Universal Robots PolyScope program: new.urp

Program new (installation=default directory=/programs/usbdisk/new folder createdIn=5.12.2.1101534 lastSavedIn=5.12.2.1101534 robotSerialNumber=20225202267)
Calibrated DH parameters: a=[0.000057, -0.560337, -0.56987, 0.000044, 0.000023, 0]; d=[0.180974, -304.223407, 295.067386, 9.330269, 0.119831, 0.115671]; alpha=[1.570416, 0.000812, 0.004616, 1.569457, -1.570316, 0]; deltaTheta=[0, -0.415128, 6.624286, 0.074029, 0.000002, -0.000001]
Robot Program (runOnlyOnce=true)
  URCap MigaWeld (Migaweld, Smooth Robotics ApS) dataModel(id_key=0, tag_version=Version1_1, enable_start_button=true, node_defined=true)
    MoveJ speed 60 deg/s, acceleration 80 deg/s^2 (useActiveTCP=false) feature=Base
      Waypoint Home_position: TCP in base x=580.944 y=-683.156 z=684.176 mm, rx=-0.0105 ry=2.8514 rz=-0.1729 rad; joints [-39.068, -105.334, -75.995, -71.646, 95.235, 51.255] deg
    Wait DigitalInput pin=digital_in[1]; digitalValue=1
    SuppressedNode
      Wait DigitalInput pin=digital_in[1]; digitalValue=1
    URCap SpeedSlider (Migaweld, Smooth Robotics ApS) dataModel(set_speed=true)
    SuppressedNode
      URCap WeldParameters (Migaweld, Smooth Robotics ApS) dataModel(processnumber=113, tackWelding=false, duo=false, current=250, isjobselected=true, seqnumber_job=1, puls=true, jobnumber=7)
    SuppressedNode
      Halt
    URCap WeldItem (Migapath, Smooth Robotics ApS) dataModel(MigaPathtitle_key=WeldItem_1)
      URCap Weld seam (Migapath, Smooth Robotics ApS) dataModel(dataModelVersion=1, programVersion=1, travelSpeed=6.0, amplitude=1.4, titleKey=Weld seam, freq=1.5)
        URCap AirPoint (Migapath, Smooth Robotics ApS) dataModel(title_key=Airpoint, jump_visible=true, pose_has_been_offset=false, Pose(key=move_pose_key, Position(key=posePosition, Length(key=X value=0.629812 unit=M), Length(key=Y value=-0.677734 unit=M), Length(key=Z value=0.186771 unit=M)), Rotation(key=poseRotation, Angle(key=RX value=-1.744823 unit=RAD), Angle(key=RY value=1.701375 unit=RAD), Angle(key=RZ value=0.596492 unit=RAD))), JointPositions(key=move_joint_key, JointPosition(key=[1], Angle(key=pos value=-0.681948 unit=RAD)), JointPosition(key=[2], Angle(key=pos value=-1.838358 unit=RAD)), JointPosition(key=[3], Angle(key=pos value=-1.393197 unit=RAD)), JointPosition(key=[4], Angle(key=pos value=-1.363283 unit=RAD)), JointPosition(key=[5], Angle(key=pos value=1.661996 unit=RAD)), JointPosition(key=[6], Angle(key=pos value=0.894606 unit=RAD))))
        URCap AirPoint (Migapath, Smooth Robotics ApS) dataModel(title_key=Startpoint, pose_has_been_offset=false, Pose(key=move_pose_key, Position(key=posePosition, Length(key=X value=0.564215 unit=M), Length(key=Y value=-0.556384 unit=M), Length(key=Z value=0.100836 unit=M)), Rotation(key=poseRotation, Angle(key=RX value=-1.592271 unit=RAD), Angle(key=RY value=1.653557 unit=RAD), Angle(key=RZ value=0.851113 unit=RAD))), JointPositions(key=move_joint_key, JointPosition(key=[1], Angle(key=pos value=-0.675332 unit=RAD)), JointPosition(key=[2], Angle(key=pos value=-1.837109 unit=RAD)), JointPosition(key=[3], Angle(key=pos value=-1.509481 unit=RAD)), JointPosition(key=[4], Angle(key=pos value=-1.463401 unit=RAD)), JointPosition(key=[5], Angle(key=pos value=1.748985 unit=RAD)), JointPosition(key=[6], Angle(key=pos value=0.902886 unit=RAD))))
        URCap Arc On (Migaweld, Smooth Robotics ApS) dataModel(arcOnWaitTime=0.0)
        URCap Paths: (Migapath, Smooth Robotics ApS)
          URCap Welding path (Migapath, Smooth Robotics ApS) dataModel(titleKey=Linear_1, selectedPathType=Linear, useShared=true, selectedPattern=ZigZag, end_has_been_offset=false, Pose(key=endPose, Position(key=posePosition, Length(key=X value=0.594829 unit=M), Length(key=Y value=-0.556361 unit=M), Length(key=Z value=0.100774 unit=M)), Rotation(key=poseRotation, Angle(key=RX value=-1.592161 unit=RAD), Angle(key=RY value=1.653589 unit=RAD), Angle(key=RZ value=0.851163 unit=RAD))), JointPositions(key=endJoint, JointPosition(key=[1], Angle(key=pos value=-0.653154 unit=RAD)), JointPosition(key=[2], Angle(key=pos value=-1.869678 unit=RAD)), JointPosition(key=[3], Angle(key=pos value=-1.467817 unit=RAD)), JointPosition(key=[4], Angle(key=pos value=-1.468622 unit=RAD)), JointPosition(key=[5], Angle(key=pos value=1.751117 unit=RAD)), JointPosition(key=[6], Angle(key=pos value=0.925296 unit=RAD))))
        URCap Arc Off (Migaweld, Smooth Robotics ApS) dataModel(arcOffWaitTime=0.5)
        URCap AirPoint (Migapath, Smooth Robotics ApS) dataModel(title_key=Airpoint, pose_has_been_offset=false, Pose(key=move_pose_key, Position(key=posePosition, Length(key=X value=0.625873 unit=M), Length(key=Y value=-0.624382 unit=M), Length(key=Z value=0.135159 unit=M)), Rotation(key=poseRotation, Angle(key=RX value=-1.620174 unit=RAD), Angle(key=RY value=1.66238 unit=RAD), Angle(key=RZ value=0.691346 unit=RAD))), JointPositions(key=move_joint_key, JointPosition(key=[1], Angle(key=pos value=-0.69265 unit=RAD)), JointPosition(key=[2], Angle(key=pos value=-1.869631 unit=RAD)), JointPosition(key=[3], Angle(key=pos value=-1.428521 unit=RAD)), JointPosition(key=[4], Angle(key=pos value=-1.387728 unit=RAD)), JointPosition(key=[5], Angle(key=pos value=1.750254 unit=RAD)), JointPosition(key=[6], Angle(key=pos value=0.925419 unit=RAD))))
    MoveJ speed 60 deg/s, acceleration 80 deg/s^2 (useActiveTCP=false) feature=Base
      Waypoint Home_position: TCP in base x=580.944 y=-683.156 z=684.176 mm, rx=-0.0105 ry=2.8514 rz=-0.1729 rad; joints [-39.068, -105.334, -75.995, -71.646, 95.235, 51.255] deg
